// TIA Portal V20 export
DATA_BLOCK "S7通信读写_1200"   // DB5
// stored: InstanceOfName S7通信读写, InstanceOfType FB
"S7通信读写"
   // VAR_INPUT
   //    连接ID : Word;
   // END_VAR
   // VAR_OUTPUT
   //    PUT_STATUS : Word;
   //    GET_STATUS : Word;
   // END_VAR
   // VAR_IN_OUT
   //    PUT_ADDR_1 : Remote;
   //    PUT_SD_1 : Variant;
   //    GET_ADDR_1 : Remote;
   //    GET_SD_1 : Variant;
   // END_VAR
   // VAR
   //    PUT_Instance { S7_SetPoint := 'True'} : PUT;
   //    GET_Instance { S7_SetPoint := 'True'} : GET;
   //    PUTdone : Bool;
   //    PUTerror : Bool;
   //    GETdone : Bool;
   //    GETerror : Bool;
   // END_VAR
BEGIN
END_DATA_BLOCK
